// Brief: Slave Arm test
FUNCTION_BLOCK PUBLIC FB_SlaveCtrlTest_1 EXTENDS FB_SlaveArmCtrlBase
VAR_INPUT
END_VAR
VAR_OUTPUT
END_VAR
VAR
	//frequency test flag	
	m_freqTestFlag :ARRAY[1..6] OF BOOL;
	
	//step test flag
	m_stepTestFlag :ARRAY[1..6] OF BOOL;
	
	//init DH joint position
	m_initDHJntPos :Vec6d;
	
	//target DH joint position
	m_targetDHJntPos :Vec6d;
	
	//target DH joint position
	m_targetDHJntVel :Vec6d;
	
	//joint motion frequency
	m_jntMotionFreq :Vec6d :=[0.2, 0.2, 0.1, 3(0.1)];
	
	//joint motion range
	m_jntMotionRange :Vec6d :=[pi/6, pi/6, 0.1, 3(pi/6)];
	
	//test joint id
	m_testJntIdx :INT :=1;	
	
	//step test joint angle
	m_jntStep : LREAL := 3*g_deg2Rad;
	
	//arm step test cycle
	m_stepCycle:LREAL:=5;
	
	//step test direction
	m_stepTestDir :ARRAY[1..6] OF INT:=[1,1,1,1,1,1];
	
	//cycle time
	m_cycleTime:LREAL:=5;
	
	//timer
	m_time:LREAL;
	
	//parameters init flag
	m_paramInitFlag,m_paramInitFlagLast:BOOL;
	
	//start motion flag
	m_startMotion,m_startMotionLast:BOOL;
	
	//test step
	m_testStep:INT:=-1;
	
	//last command position
	m_lastCmdJntPos:Vec8d;
	
	// simulated DH joint position
	m_simDHJntPos : Vec6d;
	
	// simulated slave twist of DH joint
	m_simDHJointVel :Vec6d;
	
	// commmand yaw angle and velocity
	m_cmdYawAngle :LREAL;
	m_cmdYawVel :LREAL;
	
	// instrument controller
	m_basicInstruController : FB_BasicInstruControl;
	
	// slave command grip angle and grip force level
	m_slaveCmdGripAngle :LREAL;
	m_slaveCmdGripForceLevel:LREAL;
END_VAR

METHOD armJntTest : BOOL
VAR_INPUT
	i_slaveArm :FB_SlaveArm;
END_VAR


CASE m_testStep OF 
	0://init the parameters
		m_initDHJntPos:=i_slaveArm.curDHJntPos;
		m_cmdJntPos:=i_slaveArm.curJntPos;		
		m_lastCmdJntPos:=m_cmdJntPos;
		m_cmdJntVel:=g_zeroVec8d;
		m_time:=0;
		IF (m_testJntIdx >=1 AND m_testJntIdx <=6) THEN
			m_testStep:=10;
		END_IF		
		
	
	10:// start the motion
		m_time:=m_time+g_slaveArmCtrlCycleTime;
		
		//frequency test
		IF (m_freqTestFlag[m_testJntIdx]=TRUE) THEN 
			m_targetDHJntPos[m_testJntIdx]:=m_initDHJntPos[m_testJntIdx]+m_jntMotionRange[m_testJntIdx]/2
												+0.5*m_jntMotionRange[m_testJntIdx]*SIN(2*pi*m_jntMotionFreq[m_testJntIdx]*m_time-pi/2);
			m_targetDHJntVel[m_testJntIdx]:=0.5*m_jntMotionRange[m_testJntIdx]*2*pi*m_jntMotionFreq[m_testJntIdx]*COS(2*pi*m_jntMotionFreq[m_testJntIdx]*m_time-pi/2);
		END_IF
		
		//step test
		IF (m_stepTestFlag[m_testJntIdx]=TRUE) THEN
			IF (m_time>m_cycleTime) THEN	
				m_time:=0;			
				IF (m_stepTestDir[m_testJntIdx]=1) THEN
					m_stepTestDir[m_testJntIdx]:=-1;
				ELSE
					m_stepTestDir[m_testJntIdx]:=1;
				END_IF
				//update the target joint position
				m_targetDHJntPos[m_testJntIdx]:=m_initDHJntPos[m_testJntIdx]+0.5*m_jntStep*m_stepTestDir[m_testJntIdx];
				m_targetDHJntVel[m_testJntIdx]:=0;
			END_IF		
		END_IF
		
		// calculate target motor joint position/velocity from DH joint position
		m_simDHJntPos:=m_targetDHJntPos;
		m_simDHJointVel:=m_targetDHJntVel;
		i_slaveArm.instrument.instruIK(m_targetDHJntPos,0, o_jntPos=>m_cmdJntPos);
		
		// compute command joint velocity
		vecSub(m_cmdJntPos, m_lastCmdJntPos, m_cmdJntVel);
		vecSelfMultiNum(m_cmdJntVel, g_slaveArmCtrlFreq);
		m_lastCmdJntPos:=m_cmdJntPos;
		
		//finish the test
		IF (m_startMotion=FALSE) THEN
			m_testStep:=20;
		END_IF
		
		
	20://finish signal
		m_testStep:=-1;
		
	
	-1: //
END_CASE
END_METHOD

METHOD PROTECTED calcCmdJntPos : BOOL
VAR_IN_OUT CONSTANT
	i_endoscopePose : ST_Frame;
	i_masterStatus :ST_MasterStatus;
	i_setupStatus: ST_SetupStatus;
	i_slaveArm :FB_SlaveArm;
END_VAR

VAR 
	//
END_VAR


//init parameters flag
IF (m_startMotionLast=FALSE) AND (m_startMotion=TRUE)THEN
	m_testStep:=0;
END_IF
m_startMotionLast:=m_startMotion;

//frequency test and step test
armJntTest(i_slaveArm);
END_METHOD

// override this function in each exact controller
METHOD PROTECTED calcCmdJntTrq : BOOL
VAR_IN_OUT CONSTANT
	i_endoscopePose : ST_Frame;
	i_masterStatus :ST_MasterStatus;
	i_setupStatus: ST_SetupStatus;
	i_slaveArm :FB_SlaveArm;
END_VAR

VAR 
	i:INT;
	instruCmdJntPos, instruCmdJntVel : Vec5d;	
	instruJntCtrlTrq :Vec5d;
END_VAR

// set joint torque to zero in default
m_cmdJntTrq := g_zeroVec8d;

// instrument joint control
FOR i:=1 TO 5 DO 
	instruCmdJntPos[i]:=m_cmdJntPos[i+3];
	instruCmdJntVel[i]:=m_cmdJntVel[i+3];
END_FOR
m_cmdYawAngle := m_simDHJntPos[6];
m_cmdYawVel := m_simDHJointVel[6];

m_basicInstruController.run(instruCmdJntPos,instruCmdJntVel, m_cmdYawAngle, m_cmdYawVel, m_slaveCmdGripForceLevel, i_slaveArm, o_cmdJntTrq=>instruJntCtrlTrq);
FOR i:=1 TO 5 DO
	m_cmdJntTrq[i+3]:=instruJntCtrlTrq[i];
END_FOR
END_METHOD

METHOD PUBLIC init : BOOL
VAR_IN_OUT CONSTANT
	i_slaveArm	:FB_SlaveArm;
END_VAR
VAR_IN_OUT 
	r_slaveArmCtrlCmd :ST_SlaveArmCtrlCmds;
END_VAR
SUPER^.Init(i_slaveArm,r_slaveArmCtrlCmd);

(*
m_jntOPMode[1] := DriverOPMode_PosTrq;
m_jntOPMode[2] := DriverOPMode_PosTrq;
m_jntOPMode[3] := DriverOPMode_PosTrq;
m_jntOPMode[4] := DriverOPMode_Trq;
m_jntOPMode[5] := DriverOPMode_Trq;
m_jntOPMode[6] := DriverOPMode_Trq;
m_jntOPMode[7] := DriverOPMode_Trq;
m_jntOPMode[8] := DriverOPMode_Trq;
*)

// update commands to arm
copyCmds(r_slaveArmCtrlCmd);
END_METHOD

END_FUNCTION_BLOCK

(* stored: Version 1.1.0.1, ProductVersion 3.1.4024.11
   POU FB_SlaveCtrlTest_1: Id {640a3f83-915c-4162-96a6-3f9dace817e1}, SpecialFunc None
   Method armJntTest: Id {d9baf111-002b-40c7-b14b-20ccef3a9e53}
   Method calcCmdJntPos: Id {22feec14-36e8-43db-bbdf-f70b11050ffc}
   Method calcCmdJntTrq: Id {bda90996-bd64-4dc2-a0be-75a556939603}
   Method init: Id {f2577074-2358-4a2e-9512-accf337ec1df} *)
